// TIA Portal project "Práctica 7 (sensor)" (V15)

(* hardware
DEVICE "HMI_1"  KTP700 Basic PN
   slot 0: "HMI_1"  KTP700 Basic PN  6AV2 123-2GB03-0AX0  15.0.0.0
   slot 1: "HMI_RT_1"  KTP700 Basic PN  6AV2 123-2GB03-0AX0  15.0.0.0
   slot 5: "HMI_1.IE_CP_1"  PROFINET Interface  15.0.0.0
      slot 1: "Interfaz PROFINET_1"  PROFINET Interface
         slot 1: "Port_1"  Port
DEVICE "S7-1200 station_1"  S7-1200 Station
   slot 0: "Rack_0"  S7-1200 Rack  Rack  V1.0
   slot 1: "PLC_1"  CPU 1215C AC/DC/Rly  6ES7 215-1BG40-0XB0  V4.2
*)

// ===== PLC "PLC_1"  CPU 1215C AC/DC/Rly =====

VAR_GLOBAL   // PLC tag table "Tabla de variables estándar"
   "Tag_1" AT %IW64 : Int;
   "Tag_2" AT %MD34 : DWord;
   "Tag_3" AT %MD80 : Real;
   "poco" AT %Q0.0 : Bool;
   "mucho" AT %M0.1 : Bool;
   "correcto" AT %M0.2 : Bool;
   "indicador" AT %MW3 : Int;
   "Tag_4" AT %MW100 : Word;
   "prueba" AT %MW102 : Word;
END_VAR

ORGANIZATION_BLOCK "Main"   // OB1, LAD, ProgramCycle
TITLE = "Main Program Sweep (Cycle)"
{ S7_Optimized_Access := 'TRUE' }
VERSION : 0.1
   VAR_INPUT
      Initial_Call : Bool;   // Initial call of this OB
      Remanence : Bool;   // =True, if remanent data are available
   END_VAR
BEGIN

REGION Network 1
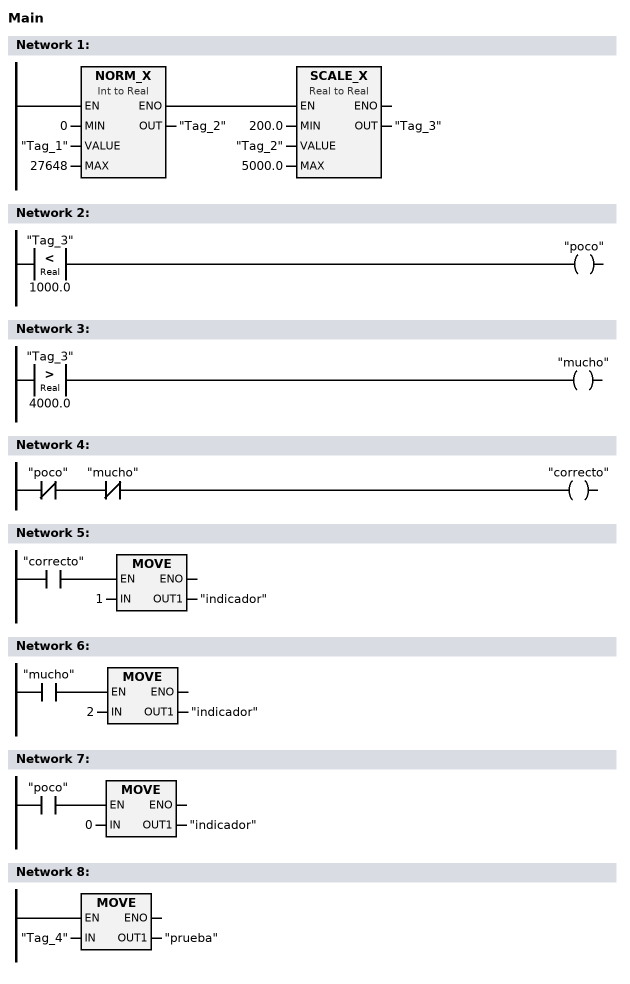
   RUNG wire#powerrail
      { S7_Templates := "[SrcType := Int, DestType := Real]" } Normalize(min := 0, value := "Tag_1", max := 27648, out => "Tag_2")
      { S7_Templates := "[SrcType := Real, DestType := Real]" } Scale(min := 200.0, value := "Tag_2", max := 5000.0, out => "Tag_3")
   END_RUNG
   // the same network as SCL:
   "Tag_2" := NORM_X(MIN := 0, VALUE := "Tag_1", MAX := 27648);
   "Tag_3" := SCALE_X(MIN := 200.0, VALUE := "Tag_2", MAX := 5000.0);
END_REGION

REGION Network 2
   RUNG wire#powerrail
      { S7_Templates := "SrcType := Real" } LT_Contact(in1 := "Tag_3", in2 := 1000.0)
      Coil( "poco" )
   END_RUNG
   // the same network as SCL:
   "poco" := "Tag_3" < 1000.0;
END_REGION

REGION Network 3
   RUNG wire#powerrail
      { S7_Templates := "SrcType := Real" } GT_Contact(in1 := "Tag_3", in2 := 4000.0)
      Coil( "mucho" )
   END_RUNG
   // the same network as SCL:
   "mucho" := "Tag_3" > 4000.0;
END_REGION

REGION Network 4
   RUNG wire#powerrail
      I_Contact( "poco" )
      I_Contact( "mucho" )
      Coil( "correcto" )
   END_RUNG
   // the same network as SCL:
   "correcto" := NOT "poco" AND NOT "mucho";
END_REGION

REGION Network 5
   RUNG wire#powerrail
      Contact( "correcto" )
      Move(in := 1, out1 => "indicador")
   END_RUNG
   // the same network as SCL:
   IF "correcto" THEN "indicador" := 1; END_IF;
END_REGION

REGION Network 6
   RUNG wire#powerrail
      Contact( "mucho" )
      Move(in := 2, out1 => "indicador")
   END_RUNG
   // the same network as SCL:
   IF "mucho" THEN "indicador" := 2; END_IF;
END_REGION

REGION Network 7
   RUNG wire#powerrail
      Contact( "poco" )
      Move(in := 0, out1 => "indicador")
   END_RUNG
   // the same network as SCL:
   IF "poco" THEN "indicador" := 0; END_IF;
END_REGION

REGION Network 8
   RUNG wire#powerrail
      Move(in := "Tag_4", out1 => "prueba")
   END_RUNG
   // the same network as SCL:
   "prueba" := "Tag_4";
END_REGION
END_ORGANIZATION_BLOCK

(* ===== HMI "HMI_RT_1" =====
connection "HMI_Conexión_1": ETHERNET, SMART_S7_1200_OMS

HMI tags "Tabla de variables estándar"
   "poco" : Bool = PLC poco AT %Q0.0, 1 s
   "indicador" : Int = PLC indicador AT %MW3, 1 s
   "prueba" : Word = PLC prueba AT %MW102, 1 s
   "Tag_3" : Real = PLC Tag_3 AT %MD80, 1 s

text list "Lista de textos_1": 0 '¡Cuidado, tanque casi vacío!'; 1 'Todo correcto.'; 2 'Tanque demasiado lleno.'

graphic list "Lista de gráficos_1": 0 'Gráfico_7'; 1 'Gráfico_8'; 2 'Gráfico_6'

graphic list "Lista de gráficos_2": 0 'Gráfico_4'; 1 'Gráfico_8'; 2 'Gráfico_9'

screen "Imagen_1" 800x480
   Visibility <- "indicador"
   Circle "Círculo_1" at 628,347 size 110x110
      Appearance <- "indicador"
   Circle "Círculo_2" at 629,109 size 109x109
      Appearance <- "indicador"
   Circle "Círculo_3" at 627,227 size 111x111
      Appearance <- "indicador"
   GraphicIOField "Campo ES gráfico_2" at 180,131 size 335x332; PictureList "Lista de gráficos_1"
      ProcessValue <- "indicador"
   TextField "Campo de texto_1" at 580,298 size 16x23; Text 'Text'
   IOField "Campo ES_1" at 186,61 size 333x55; FormatPattern s999999999.999
      ProcessValue <- "Tag_3"
   TextField "Campo de texto_2" at 186,26 size 138x23; Text 'Volumen tanque'
   Bar "Barra_1" at 22,50 size 138x407; MinimumValue 200; MaximumValue 5000
      ProcessValue <- "Tag_3"
   SymbolicIOField "Campo ES simbólico_1" at 533,16 size 248x77; TextOff '0'; TextOn '1'; TextList "Lista de textos_1"
      ProcessValue <- "indicador"
*)